// TIA Portal V18 export
// export: Created 2026-06-11T03:43:50.4308411Z, ExportSetting WithDefaults, DisplayName Totally Integrated Automation Portal, DisplayVersion V18, DisplayName TIA Portal Openness, DisplayVersion V18, DisplayName TIA Portal Version Control Interface, DisplayVersion V18, DisplayName STEP 7 Professional, DisplayVersion V18, DisplayName STEP 7 Safety, DisplayVersion V18, DisplayName WinCC Professional, DisplayVersion V18
Screen "05_Canh_Bao_IO"  800x600, Number=5
  ScreenLayer 
    GraphicView "Graphic view_1" at 0,0 size 800x600  Picture=ChatGPT Image 10_30_37 30 thg 5, 2026
    Button "Button_1" at 27,546 size 107x46  Mode=Text, TextOff="TỔNG QUAN", TextOn="Text"
      on Click: ActivateScreen(Screen name := 01_Tong_Quan, Object number := 0)
    Button "Button_2" at 153,546 size 107x46  Mode=Text, TextOff="VẬN HÀNH", TextOn="Text"
      on Click: ActivateScreen(Screen name := 02_Van_Hanh, Object number := 0)
    Button "Button_3" at 281,546 size 107x46  Mode=Text, TextOff="PID MỨC", TextOn="Text"
      on Click: ActivateScreen(Screen name := 03_PID_Muc_Nuoc, Object number := 0)
    Button "Button_4" at 409,545 size 107x46  Mode=Text, TextOff="TREND", TextOn="Text"
      on Click: ActivateScreen(Screen name := 04_Trend, Object number := 0)
    TextField "Text field_1" at 254,5 size 259x31  Text="MÀN HÌNH 05 - ALARM"
    Rectangle "Rectangle_8" at 533,542 size 114x52
    Button "Button_5" at 537,545 size 107x46  Mode=Text, TextOff="CẢNH BÁO", TextOn="Text"
      on Click: ActivateScreen(Screen name := , Object number := 0)
    Button "Button_6" at 732,554 size 65x30  Mode=Text, TextOff="EXIT", TextOn="Text"
      on Click: StopRuntime(Mode := 0)
    Rectangle "Rectangle_1" at 511,360 size 59x27
    Rectangle "Rectangle_2" at 511,407 size 59x27
    Rectangle "Rectangle_3" at 511,454 size 59x27
    Rectangle "Rectangle_4" at 703,359 size 55x28
    Rectangle "Rectangle_5" at 703,406 size 55x29
    Rectangle "Rectangle_6" at 703,453 size 56x30
    Rectangle "Rectangle_7" at 703,498 size 55x30
    Circle "Circle_1" at 44,83 size 29x29
      RangeAppearanceAnimation "RangeAppearanceAnimation"
        tag Canh_Bao_Muc_Cao
        0..0: back #c0c0c0, fore #181c31
        1..1: back #ffff00, fore #181c31
    Circle "Circle_2" at 44,127 size 29x29
      RangeAppearanceAnimation "RangeAppearanceAnimation"
        tag Canh_Bao_Muc_Thap
        0..0: back #d9d9d9, fore #181c31
        1..1: back #ffff00, fore #181c31
    Circle "Circle_3" at 44,172 size 29x29
      RangeAppearanceAnimation "RangeAppearanceAnimation"
        tag Canh_Bao_Nhiet_Cao
        0..0: back #d9d9d9, fore #181c31
        1..1: back #ffff00, fore #181c31
    Circle "Circle_4" at 44,217 size 29x29
      RangeAppearanceAnimation "RangeAppearanceAnimation"
        tag Canh_Bao_Ap_Cao
        0..0: back #d9d9d9, fore #181c31
        1..1: back #ffff00, fore #181c31
    Circle "Circle_5" at 48,338 size 22x22
      RangeAppearanceAnimation "RangeAppearanceAnimation"
        tag Loi_Muc_Cao
        0..0: back #d9d9d9, fore #181c31
        1..1: back #ff0000, fore #181c31, flashing
    Circle "Circle_6" at 48,379 size 22x22
      RangeAppearanceAnimation "RangeAppearanceAnimation"
        tag Loi_Nhiet_Cao
        0..0: back #d9d9d9, fore #181c31
        1..1: back #ff0000, fore #181c31, flashing
    Circle "Circle_7" at 48,420 size 22x22
      RangeAppearanceAnimation "RangeAppearanceAnimation"
        tag Loi_Ap_Cao
        0..0: back #d9d9d9, fore #181c31
        1..1: back #ff0000, fore #181c31, flashing
    Circle "Circle_8" at 47,458 size 25x25
      RangeAppearanceAnimation "RangeAppearanceAnimation"
        tag Nut_EStop_HMI
        0..0: back #00ff00, fore #181c31
        1..1: back #ff0000, fore #181c31, flashing
    Circle "Circle_9" at 48,499 size 22x22
      RangeAppearanceAnimation "RangeAppearanceAnimation"
        tag Loi_He_Thong
        0..0: back #d9d9d9, fore #181c31
        1..1: back #ff0000, fore #181c31, flashing
    Circle "Circle_10" at 414,103 size 29x29
      RangeAppearanceAnimation "RangeAppearanceAnimation"
        tag Nut_Start
        0..0: back #d9d9d9, fore #181c31
        1..1: back #00ff00, fore #181c31
    Circle "Circle_11" at 414,147 size 29x29
      RangeAppearanceAnimation "RangeAppearanceAnimation"
        tag Nut_Stop
        0..0: back #d9d9d9, fore #181c31
        1..1: back #ff0000, fore #181c31
    Circle "Circle_12" at 414,191 size 29x29
      RangeAppearanceAnimation "RangeAppearanceAnimation"
        tag Nut_EStop
        0..0: back #ff0000, fore #181c31
        1..1: back #00ff00, fore #181c31
    Circle "Circle_13" at 414,235 size 29x29
      RangeAppearanceAnimation "RangeAppearanceAnimation"
        tag Nut_Boiler_Ready
        0..0: back #d9d9d9, fore #181c31
        1..1: back #00ff00, fore #181c31
    Circle "Circle_14" at 593,102 size 29x29
      RangeAppearanceAnimation "RangeAppearanceAnimation"
        tag Den_Running
        0..0: back #d9d9d9, fore #181c31
        1..1: back #00ff00, fore #181c31
    Circle "Circle_15" at 593,147 size 29x29
      RangeAppearanceAnimation "RangeAppearanceAnimation"
        tag Van_Cap_Hoi
        0..0: back #d9d9d9, fore #181c31
        1..1: back #ff6600, fore #181c31
    Circle "Circle_16" at 593,191 size 29x29
      RangeAppearanceAnimation "RangeAppearanceAnimation"
        tag Bom_Lam_Mat
        0..0: back #d9d9d9, fore #181c31
        1..1: back #00ffff, fore #181c31
    Circle "Circle_17" at 593,235 size 29x29
      RangeAppearanceAnimation "RangeAppearanceAnimation"
        tag Coi_Alarm
        0..0: back #d9d9d9, fore #181c31
        1..1: back #ff0000, fore #181c31, flashing
    IOField "I/O field_8" at 516,362 size 49x24  DataFormat=Decimal, FormatPattern=99999, Mode=Output
      ProcessValue := Muc_Nuoc_Raw
    IOField "I/O field_1" at 516,409 size 49x24  DataFormat=Decimal, FormatPattern=99999, Mode=Output
      ProcessValue := Nhiet_Do_Raw
    IOField "I/O field_2" at 516,455 size 49x24  DataFormat=Decimal, FormatPattern=99999, Mode=Output
      ProcessValue := Ap_Suat_Raw
    IOField "I/O field_3" at 707,362 size 49x24  DataFormat=Decimal, FormatPattern=9.9, Mode=Output
      ProcessValue := Muc_Nuoc_PV
    IOField "I/O field_4" at 707,410 size 49x24  DataFormat=Decimal, FormatPattern=99.9, Mode=Output
      ProcessValue := Nhiet_Do_PV
    IOField "I/O field_5" at 706,457 size 49x24  DataFormat=Decimal, FormatPattern=99.9, Mode=Output
      ProcessValue := Ap_Suat_PV
    IOField "I/O field_6" at 706,501 size 49x24  DataFormat=Decimal, FormatPattern=99999, Mode=Output
      ProcessValue := Van_Xa_Raw
